FUNCTION_BLOCK derived2 EXTENDS base implements itf
VAR_INPUT
END_VAR
VAR_OUTPUT
END_VAR
VAR
END_VAR

METHOD ITF_METH : STRING
VAR_INPUT
END_VAR
ITF_METH := 'derived2 itf method';
END_METHOD

METHOD METH : string
VAR_INPUT
END_VAR
METH := 'derived2';
END_METHOD

END_FUNCTION_BLOCK

(* stored: Version 1.1.0.1, ProductVersion 3.1.4022.10
   POU derived2: Id {97ebf8f7-b506-4f0c-841b-341e4c343500}, SpecialFunc None
   Method ITF_METH: Id {0ed03664-ab68-49eb-ab7a-5edb4057c1d9}
   Method METH: Id {c2704ac9-6f41-43a1-83e2-29aada0b9573} *)
